PROGRAM Stn051_26_Stn090MainMergePrestop
VAR
//correct
	{attribute 'TcLinkToOSO' := '.iPuckPresent    :=  <0,1,2>TIIB[N23S00 (AL1332)]^N23S01 (AL2341)^TxPDO^input byte 1;
		.iBufferFull  :=  <0,1,2>TIIB[N23S00 (AL1332)]^N23S01 (AL2341)^TxPDO^input byte 3;
		.oStopLower   :=  <0,1,1>TIIB[N24S00 (AL1332)]^N24S02 (EX260)^RxPDO^output byte 0'}
	fbConvStop: FB_ConvStop;
END_VAR

//  This code instantiates a component that is implimented as a common function block
//    Note that I/O is linked directly to I/O variables inside the named instance

gStn051_26_Stn090MainMergePrestop.ConvRunning  := gConsumed_SafetyInterfaceConv.MtrRunning.Enc053Mtr04;

fbConvStop(
	pStn := ADR(gStn051),
	pCmp := ADR(gStn051_26_Stn090MainMergePrestop),
	pUpstreamStop := 0,
	pStateTraceBuffer := ADR(gStn051_StateTraceBuffer),
	pStateTraceFifo := ADR(gStn051_StateTraceFifo),
	pStats := ADR(gStn051_02_Stats));

END_PROGRAM

(* stored: Version 1.1.0.1, ProductVersion 3.1.4024.6
   POU Stn051_26_Stn090MainMergePrestop: Id {dda19376-088f-4be3-a214-537b9b386d20}, SpecialFunc None *)
